FUNCTION_BLOCK CentralServer
  (* Standard: 61499-2 *)
  (* Version 0.2, 2003-12-04, JHC, Rockwell Automation, Renamed for better indexing. *)
  (* Version 0.1, 2002-11-05, JHC, Rockwell Automation, Corrected missing ST element in Algorithm REQ. *)
  (* Version 0.0, 2000-05-30, JHC, Rockwell Automation *)
  (* Compiler header: package fb.rt.cs725; *)
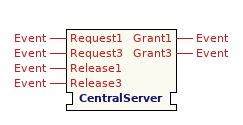
  EVENT_INPUT
    Request1; (* Initialization Request *)
    Request3; (* dab *)
    Release1;
    Release3;
  END_EVENT
  EVENT_OUTPUT
    Grant1; (* Initialization Confirm *)
    Grant3; (* Execution Confirmation *)
  END_EVENT
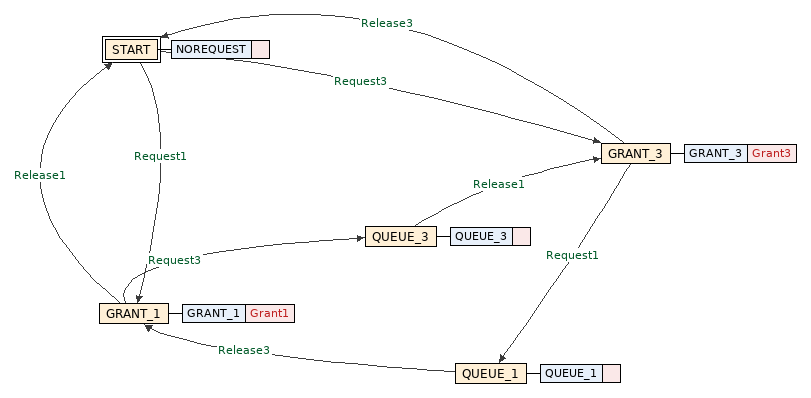
  EC_STATES
    START : NOREQUEST; (* Init state *)
    GRANT_1 : GRANT_1 -> Grant1;
    GRANT_3 : GRANT_3 -> Grant3;
    QUEUE_3 : QUEUE_3;
    QUEUE_1 : QUEUE_1;
  END_STATES
  EC_TRANSITIONS
    START TO GRANT_1 := Request1;
    GRANT_1 TO START := Release1;
    START TO GRANT_3 := Request3;
    GRANT_3 TO START := Release3;
    GRANT_1 TO QUEUE_3 := Request3;
    QUEUE_3 TO GRANT_3 := Release1;
    GRANT_3 TO QUEUE_1 := Request1;
    QUEUE_1 TO GRANT_1 := Release3;
  END_TRANSITIONS
  ALGORITHM GRANT_1 IN Java: (* Initialization algorithm *)
System.out.println("Token granted to FC1");
  END_ALGORITHM
  ALGORITHM GRANT_3 IN Java: (* Initialization algorithm *)
System.out.println("Token granted to FC3");
  END_ALGORITHM
  ALGORITHM NOREQUEST IN Java: (* Normally executed algorithm *)
System.out.println("No request");
  END_ALGORITHM
  ALGORITHM QUEUE_3 IN Java: (* Normally executed algorithm *)
System.out.println("FC3 waiting for token");
  END_ALGORITHM
  ALGORITHM QUEUE_1 IN Java: (* Normally executed algorithm *)
System.out.println("FC1 waiting for token");
  END_ALGORITHM
END_FUNCTION_BLOCK
